(* CODESYS project SP16FlightSimPLC.export

Project tree, tasks and I/O mapping:
  Device : EHV-CPU1025, Hitachi-IES, order no. EHV-CPU1025, version 3.5.4.11
    application Application
      libraries: Standard, * (System); SysTimeRtc, 3.5.17.0 (System); CAA Net Base Services, 3.5.8.10 (CAA Technical Workgroup); PRO JSON, 1.0.0.11 (Pro Electric)
      task MainTask (cyclic, interval 20 ms, priority 1) calls TcpClient
      data type ServoData
      global variables GVL
      global variables gvlSetting
      program TcpClient [ST]
    Basic : Basic, Hitachi-IES, version 3.4.4.0
      <Empty>
      <Empty>
      <Empty>
      <Empty>
      <Empty>
      <Empty>
      <Empty>
      <Empty>
      <Empty>
      <Empty>
      <Empty>
*)

// Device/Application/ServoData
TYPE ServoData :
STRUCT
	positions: ARRAY[1..6] OF JSONVAR;
	speeds: ARRAY[1..6] OF JSONVAR;
END_STRUCT
END_TYPE

// Device/Application/GVL
{attribute 'qualified_only'}
VAR_GLOBAL
    sIpAddr    :    NBS.IP_ADDR := (sAddr := '145.48.203.188'); // Change to own IP-Address
    // !!!  Make sure that the firewall does not block these ports !!!
    uiPort     :    UINT := 51223; // Port for the sender => receiver will set to uiPort + 1
END_VAR

// Device/Application/gvlSetting
{attribute 'qualified_only'}
VAR_GLOBAL CONSTANT
    gc_uiPort        : UINT := 51223;
    gc_stIpAddr      : NBS.IP_ADDR := (sAddr := '145.48.203.188');
     
    gc_wMaxTelegram  : INT := 250; // Length o the telegram
END_VAR

// Device/Application/TcpClient
PROGRAM TcpClient
VAR
    fbTcpClient   : NBS.TCP_Client;
    fbTcpRead     : NBS.TCP_Read;
    fbTcpWrite    : NBS.TCP_Write;
 
    abyTx         : ARRAY [0..gvlSetting.gc_wMaxTelegram] OF BYTE;
    abyRx         : ARRAY [0..gvlSetting.gc_wMaxTelegram] OF BYTE;
	received      : STRING(gvlSetting.gc_wMaxTelegram);
	sent          : STRING(gvlSetting.gc_wMaxTelegram);
	parseJSON     : JSON_TO_STRUCT;
	composeJSON   : STRUCT_TO_JSON;
	servoData     : ServoData;
 
    udiVal        : UDINT;
    pudiVal       : POINTER TO BYTE;
    iIndex        : INT;
    xConnect      : BOOL;
 
    xRead         : BOOL := TRUE;
    xMissingAck   : BOOL;
    udiResult     : UDINT;
    udiLastAck    : UDINT;
    udiNow        : UDINT;
    udiRead       : UDINT;
END_VAR

fbTcpClient(xEnable := xConnect, ipAddr := gvlSetting.gc_stIpAddr, uiPort := gvlSetting.gc_uiPort, udiTimeOut := 0);

composeJSON(
	Execute:= TRUE,
	JSONString:= ADR(sent), 
	JSONStringSize:= SIZEOF(sent),
	JSONVars:= ADR(servoData.positions),
	NumberOfVars:= SIZEOF(servoData.positions) / SIZEOF(JSONVAR)
);

composeJSON(Execute:= FALSE);

fbTcpWrite(xExecute := xConnect, hConnection := fbTcpClient.hConnection, udiTimeOut := 0, szSize := SIZEOF(sent), pData := ADR(sent));
fbTcpWrite(xExecute := FALSE);


fbTcpRead(xEnable := xRead AND xConnect, hConnection := fbTcpClient.hConnection, szSize := SIZEOF(received), pData := ADR(received), szCount => udiRead);
 
parseJSON(	
	Execute := TRUE,
    JSONString:= ADR(received), 
    JSONStringSize:= SIZEOF(received),
    JSONVars:= ADR(servoData),
    NumberOfVars:= SIZEOF(servoData) / SIZEOF(JSONVAR)
);
parseJSON(Execute:= FALSE);

IF fbTcpRead.xError THEN
    fbTcpRead(xEnable := FALSE);
END_IF
 
IF NOT fbTcpClient.xActive AND NOT fbTcpClient.xBusy AND NOT fbTcpClient.xDone THEN
    xConnect := TRUE;
ELSIF fbTcpClient.xDone THEN
    xConnect := FALSE;
END_IF

END_PROGRAM
